SYSTEM ControlPanel (* System Configuration *)
  (* Standard: 61499-1 *)
  (* Version 0.3, 2003-12-05, JHC, Rockwell Automation, Renamed from NEWSYSTEM. *)
  (* Version 0.2, 2002-11-05, JHC, Rockwell Automation, Fixed missing (empty) FBD in Application. *)
  (* Version 0.1, 2002-01-17, JHC, Rockwell Automation, Minor cleanup *)
  (* Version 0.0, 2000-05-27, JHC, Rockwell Automation *)
  APPLICATION APP1
  END_APPLICATION
  DEVICE WorkerHMI : FRAME_DEVICE(BOUNDS := [500,300,300,300], GRID := [1,1])
    RESOURCE Worker_1_HMI : PANEL_RESOURCE(ROWS := 4, COLS := 2)
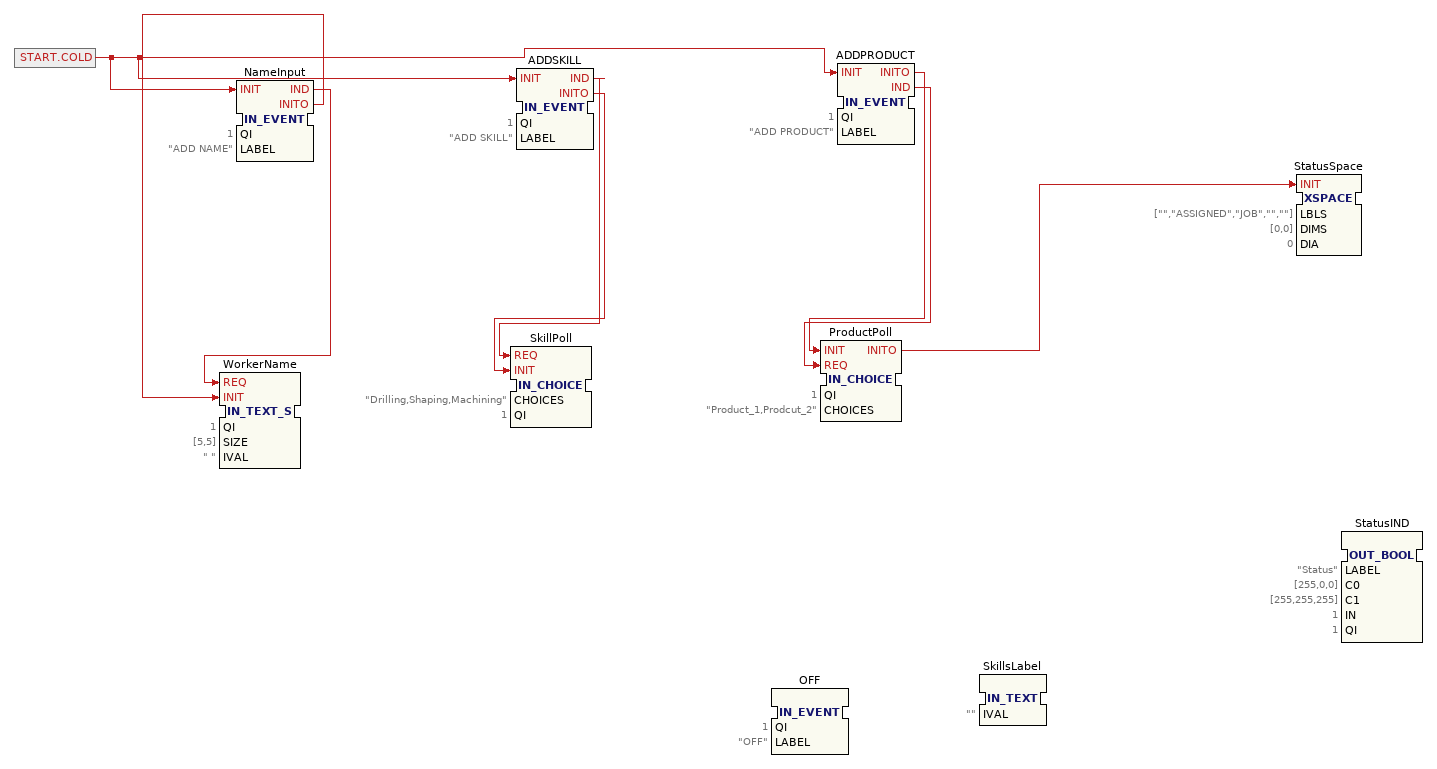
      FBS
        NameInput : IN_EVENT(QI := 1, LABEL := "ADD NAME");
        SkillPoll : IN_CHOICE(CHOICES := "Drilling,Shaping,Machining", QI := 1);
        StatusIND : OUT_BOOL(LABEL := "Status", C0 := [255,0,0], C1 := [255,255,255], IN := 1, QI := 1);
        OFF : IN_EVENT(QI := 1, LABEL := "OFF");
        SkillsLabel : IN_TEXT(IVAL := "");
        ADDSKILL : IN_EVENT(QI := 1, LABEL := "ADD SKILL");
        WorkerName : IN_TEXT_S(QI := 1, SIZE := [5,5], IVAL := "    ");
        ProductPoll : IN_CHOICE(QI := 1, CHOICES := "Product_1,Prodcut_2");
        ADDPRODUCT : IN_EVENT(QI := 1, LABEL := "ADD PRODUCT");
        StatusSpace : XSPACE(LBLS := ["","ASSIGNED","JOB","",""], DIMS := [0,0], DIA := 0);
      END_FBS
      EVENT_CONNECTIONS
        START.COLD TO NameInput.INIT;
        ADDSKILL.IND TO SkillPoll.REQ;
        ADDSKILL.INITO TO SkillPoll.INIT;
        NameInput.IND TO WorkerName.REQ;
        START.COLD TO ADDSKILL.INIT;
        NameInput.INITO TO WorkerName.INIT;
        ADDPRODUCT.INITO TO ProductPoll.INIT;
        ADDPRODUCT.IND TO ProductPoll.REQ;
        START.COLD TO ADDPRODUCT.INIT;
        ProductPoll.INITO TO StatusSpace.INIT;
      END_CONNECTIONS
    END_RESOURCE
  END_DEVICE
END_SYSTEM
